(* IEC 61131-3 sources: Lasal/CPU_5344_V01/Class/cmToolChange, 1 file *)

(* ---- cmToolChange.st ---- *)
(*!
<Class
	Name               = "cmToolChange"
	Revision           = "0.0"
	RealtimeTask       = "false"
	CyclicTask         = "true"
	DefCyclictime      = "10 ms"
	BackgroundTask     = "true"
	Sigmatek           = "false"
	OSInterface        = "false"
	HighPriority       = "false"
	Automatic          = "false"
	UpdateMode         = "Prescan"
	SharedCommandTable = "true"
	Objectsize         = "(450,720)">
	<Channels>
		<Server Name="iSimuChange" Visualized="false" Initialize="false" WriteProtected="false" Retentive="false"/>
		<Server Name="oToolOk" Visualized="false" Initialize="false" WriteProtected="true" Retentive="false"/>
		<Server Name="parWaitTimeForBlowCoin" Visualized="true" Initialize="true" DefValue="1000" WriteProtected="false" Retentive="File"/>
		<Server Name="stprChange" Visualized="false" Initialize="false" WriteProtected="false" Retentive="false"/>
		<Client Name="iCmdToolChange" Required="true" Internal="false"/>
		<Client Name="iMotorStandStill" Required="true" Internal="false"/>
		<Client Name="iNoTool" Required="true" Internal="false"/>
		<Client Name="iToolLocked" Required="true" Internal="false"/>
		<Client Name="oBlowCone" Required="true" Internal="false"/>
		<Client Name="oChangeTool" Required="true" Internal="false"/>
	</Channels>
	<Network Name="cmToolChange">
		<!-- List of Components in this network -->
		<Components>
			<Object
				Name       = "_base"
				Class      = "cmBase"
				Position   = "(218,120)"
				Visualized = "true">
				<Channels>
					<Server Name="ClassSvr"/>
					<Server Name="cmdHMI"/>
					<Server Name="ErrorNr"/>
					<Server Name="mode"/>
					<Server Name="state"/>
					<Server Name="stsHMI_RunsAllowed"/>
					<Server Name="stsInAlarm"/>
					<Server Name="stsIsInterlocked"/>
					<Client Name="id"/>
					<Client Name="nwEmOrUnit"/>
				</Channels>
			</Object>
		</Components>
		<Comments>
		</Comments>
		<!-- List of Connections in this network -->
		<Connections>
			<Connection Source="this.ClassSvr" Destination="_base.ClassSvr" Vertices="(1036,210),(864,210),"/>
			<Connection Source="this.state" Destination="_base.state" Vertices="(1036,270),(864,270),"/>
			<Connection Source="this.mode" Destination="_base.mode" Vertices="(1036,330),(864,330),"/>
			<Connection Source="this.cmdHMI" Destination="_base.cmdHMI" Vertices="(1036,390),(864,390),"/>
			<Connection Source="this.stsInAlarm" Destination="_base.stsInAlarm" Vertices="(1036,450),(864,510),"/>
			<Connection Source="this.stsIsInterlocked" Destination="_base.stsIsInterlocked" Vertices="(1036,510),(864,570),"/>
			<Connection Source="this.stsHMI_RunsAllowed" Destination="_base.stsHMI_RunsAllowed" Vertices="(1036,570),(864,630),"/>
			<Connection Source="this.ErrorNr" Destination="_base.ErrorNr" Vertices="(1036,630),(864,690),"/>
			<Connection Source="_base.nwEmOrUnit" Destination="this.nwEmOrUnit" Vertices="(218,210),(38,210),"/>
			<Connection Source="_base.id" Destination="this.id" Vertices="(218,270),(38,270),"/>
		</Connections>
		<!-- Headerfiles -->
		<Options>
		</Options>
	</Network>
</Class>
*)
#pragma using cmBase

cmToolChange : CLASS
: cmBase
  //Servers:
	parWaitTimeForBlowCoin 	: SvrCh_UDINT;
	stprChange 	: SvrCh_DINT;
	iSimuChange 	: SvrCh_DINT;
	oToolOk 	: SvrCh_DINT;
  //Clients:
	iNoTool 	: CltCh_DINT;
	iMotorStandStill 	: CltCh_DINT;
	iToolLocked 	: CltCh_DINT;
	iCmdToolChange 	: CltCh_DINT;
	oChangeTool 	: CltCh_DINT;
	oBlowCone 	: CltCh_DINT;
  //Variables:
		oldCmdToolChange 	: DINT;
		timerWaitForBlowCoin 	: strTimer;
  //Functions:

	FUNCTION VIRTUAL work;

	FUNCTION VIRTUAL preScanOverride;

	FUNCTION VIRTUAL postScanOverride;
  //Tables:
	FUNCTION @STD
		VAR_OUTPUT
			ret_code	: CONFSTATES;
		END_VAR;
	FUNCTION GLOBAL TAB @CT_;
END_CLASS;

// JdK 3-10-2019 cm tool change, created for 4255 and standard lib
// task of this cm is to control the toolchange, and to check if tool is ok

// toolchange is only allowed if state is aborted
// there are no errors

FUNCTION VIRTUAL cmToolChange::work

  CASE stprChange OF

  0: //wait for command
    IF pmlCom.cmd.state= Aborted & iCmdToolChange= 1 & oldCmdToolChange= 1 & iMotorStandStill= 1 THEN //only on positive trigger
      stprChange+= 1;
    END_IF;

  1: //set change tool output to 1, wait for blow coin output
    oChangeTool:=1;
    IF timerWaitForBlowCoin.done THEN
      stprChange+=1;
    END_IF;

  2: //set both outputs to 1
    oChangeTool:= 1;
    oBlowCone:= 1;

  END_CASE;

END_FUNCTION

FUNCTION VIRTUAL cmToolChange::preScanOverride

  //read inputs
  IF pmlCom.cmd.simulation <> allSimu THEN
    iNoTool := iNoTool.Read();
    iMotorStandStill := iMotorStandStill.Read();
    iToolLocked := iToolLocked.Read();
    iCmdToolChange:= iCmdToolChange.Read();
  ELSE //simulations, set all to ok values
    iNoTool:= 0;
    iMotorStandStill:= 1;
    iToolLocked:= 1;
    iCmdToolChange:= iSimuChange;
  END_IF;

  //always set outputs to 0, if required they are in work set to a value
  oChangeTool:= 0;
  oBlowCone:= 0;

  //stop toolchange if no longer aborted
  IF pmlCom.cmd.state <> Aborted | iCmdToolChange= 0 THEN
    stprChange:= 0; //always stop if state isn't aborted
  END_IF;

  //run timer wait for blow
  timerWaitForBlowCoin:= runTimer(Active:=stprChange=1, iMem:=timerWaitForBlowCoin, TimerTime:=parWaitTimeForBlowCoin, Pause:=0);

END_FUNCTION

FUNCTION VIRTUAL cmToolChange::postScanOverride

  //write outputs
  oToolOk:=iNoTool=0 & iToolLocked= 1 & oChangeTool=0 & oBlowCone=0 ;
  oChangeTool.Write(input:=oChangeTool);
  oBlowCone.Write(input:=oBlowCone);

  //set trigger merker
  oldCmdToolChange:= iCmdToolChange;

END_FUNCTION
